% RSLogix 500 project P5_ABIOLA_A_BAK060.RSS, saved by version 8.30.00.16 %
PROJECT "UNTITLED"    % processor: Bul.1763 MicroLogix 1100 Series B %

PROGRAM FILES
  LAD 2   6 rungs
  LAD 3 "I/O"  1 rungs  % This contains all the input and output logic %

DATA FILES
  O0 OUTPUT  4 elements
  I1 INPUT  6 elements
  S2 STATUS  66 elements
  B3 BINARY  1 elements
  T4 TIMER  3 elements
  C5 COUNTER  2 elements
  R6 CONTROL  1 elements
  N7 INTEGER  1 elements
  F8 FLOAT  2 elements

LADDER 2
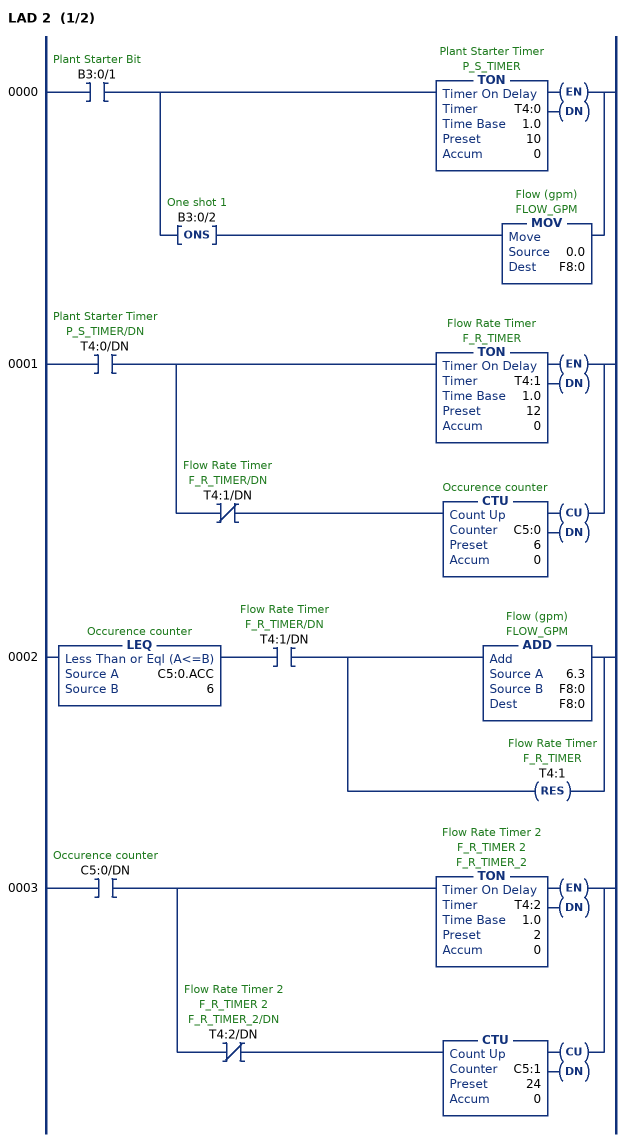
% Rung: 0 %
SOR XIC B3:0/1 BST TON T4:0 1.0 10 0 NXB ONS B3:0/2 MOV 0.0 F8:0 BND EOR
%   B3:0/1  "Plant Starter Bit" %
%   T4:0  P_S_TIMER  "Plant Starter Timer" %
%   B3:0/2  "One shot 1" %
%   F8:0  FLOW_GPM  "Flow (gpm)" %
% Rung: 1 %
SOR XIC T4:0/DN BST TON T4:1 1.0 12 0 NXB XIO T4:1/DN CTU C5:0 6 0 BND EOR
%   T4:0  P_S_TIMER  "Plant Starter Timer" %
%   T4:1  F_R_TIMER  "Flow Rate Timer" %
%   C5:0  "Occurence counter" %
% Rung: 2 %
SOR LEQ C5:0.ACC 6 XIC T4:1/DN BST ADD 6.3 F8:0 F8:0 NXB RES T4:1 BND EOR
%   C5:0  "Occurence counter" %
%   T4:1  F_R_TIMER  "Flow Rate Timer" %
%   F8:0  FLOW_GPM  "Flow (gpm)" %
% Rung: 3 %
SOR XIC C5:0/DN BST TON T4:2 1.0 2 0 NXB XIO T4:2/DN CTU C5:1 24 0 BND EOR
%   C5:0  "Occurence counter" %
%   T4:2  F_R_TIMER_2  "Flow Rate Timer 2 F_R_TIMER 2" %

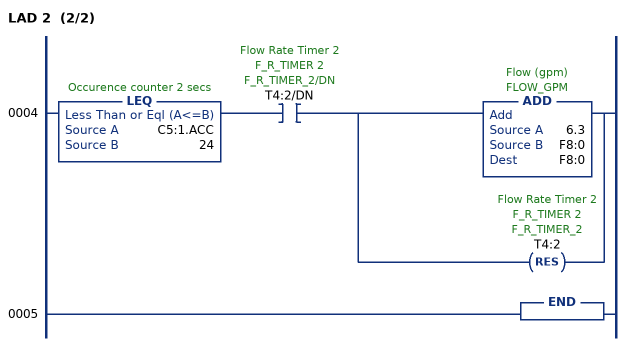
% Rung: 4 %
SOR LEQ C5:1.ACC 24 XIC T4:2/DN BST ADD 6.3 F8:0 F8:0 NXB RES T4:2 BND EOR
%   C5:1.ACC  "Occurence counter 2 secs" %
%   T4:2  F_R_TIMER_2  "Flow Rate Timer 2 F_R_TIMER 2" %
%   F8:0  FLOW_GPM  "Flow (gpm)" %
% Rung: 5 %
SOR END EOR

OTHER DOCUMENTED ADDRESSES
  B3:0/3  "One shot 2"
  F8:1  F_R_SUM  "Flow Rate Sum"

DATA TABLE (non-zero values as saved)
DATA T4
% .PRE .ACC %
% T4:0 % 10 0
% T4:1 % 12 0
% T4:2 % 2 0
DATA C5
% .PRE .ACC %
% C5:0 % 6 0
% C5:1 % 24 0
